(* PLC project Robin, CODESYS CODESYS V3.5 SP15, author pdcribeiro *)
(* stored: creationDateTime 2019-12-17T11:46:08.0055698, version 0.1.2, modificationDateTime 2019-12-17T11:45:59.136833, organization INESC TEC *)
(* A ROS-CODESYS shared memory bridge that maps CODESYS variables to ROS topics.

https://github.com/ScalABLE40/robin *)

(* {attribute 'pack_mode' := '0'} *)
TYPE Accel : STRUCT
  linear : Vector3;
  angular : Vector3;
END_STRUCT;
END_TYPE

(* {attribute 'pack_mode' := '0'} *)
TYPE AccelStamped : STRUCT
  header : Header;
  accel : Accel;
END_STRUCT;
END_TYPE

(* {attribute 'pack_mode' := '0'} *)
TYPE AccelWithCovariance : STRUCT
  accel : Accel;
  covariance : ARRAY[1..36] OF LREAL;
END_STRUCT;
END_TYPE

(* {attribute 'pack_mode' := '0'} *)
TYPE AccelWithCovarianceStamped : STRUCT
  header : Header;
  accel : AccelWithCovariance;
END_STRUCT;
END_TYPE

(* {attribute 'pack_mode' := '0'} *)
TYPE Inertia : STRUCT
  m : LREAL;
  com : Vector3;
  ixx : LREAL;
  ixy : LREAL;
  ixz : LREAL;
  iyy : LREAL;
  iyz : LREAL;
  izz : LREAL;
END_STRUCT;
END_TYPE

(* {attribute 'pack_mode' := '0'} *)
TYPE InertiaStamped : STRUCT
  header : Header;
  inertia : Inertia;
END_STRUCT;
END_TYPE

(* /{attribute 'pack_mode' := '0'} *)
TYPE Point : STRUCT
  x : LREAL;
  y : LREAL;
  z : LREAL;
END_STRUCT;
END_TYPE

(* {attribute 'pack_mode' := '0'} *)
TYPE Point32 : STRUCT
  x : REAL;
  y : REAL;
  z : REAL;
END_STRUCT;
END_TYPE

(* {attribute 'pack_mode' := '0'} *)
TYPE PointStamped : STRUCT
  header : Header;
  point : Point;
END_STRUCT;
END_TYPE

(* {attribute 'pack_mode' := '0'} *)
TYPE Polygon : STRUCT
  {attribute 'robin_var_len'}
  points : ARRAY[1..Robin.DEF_ARRAY_LEN] OF Point32;
END_STRUCT;
END_TYPE

(* {attribute 'pack_mode' := '0'} *)
TYPE PolygonStamped : STRUCT
  header : Header;
  polygon : Polygon;
END_STRUCT;
END_TYPE

(* {attribute 'pack_mode' := '0'} *)
TYPE Pose : STRUCT
  position : Point;
  orientation : Quaternion;
END_STRUCT;
END_TYPE

(* {attribute 'pack_mode' := '0'} *)
TYPE Pose2D : STRUCT
  x : LREAL;
  y : LREAL;
  theta : LREAL;
END_STRUCT;
END_TYPE

(* {attribute 'pack_mode' := '0'} *)
TYPE PoseArray : STRUCT
  header : Header;
  {attribute 'robin_var_len'}
  poses : ARRAY[1..Robin.DEF_ARRAY_LEN] OF Pose;
END_STRUCT;
END_TYPE

(* {attribute 'pack_mode' := '0'} *)
TYPE PoseStamped : STRUCT
  header : Header;
  pose : Pose;
END_STRUCT;
END_TYPE

(* {attribute 'pack_mode' := '0'} *)
TYPE PoseWithCovariance : STRUCT
  pose : Pose;
  covariance : ARRAY[1..36] OF LREAL;
END_STRUCT;
END_TYPE

(* {attribute 'pack_mode' := '0'} *)
TYPE PoseWithCovarianceStamped : STRUCT
  header : Header;
  pose : PoseWithCovariance;
END_STRUCT;
END_TYPE

(* {attribute 'pack_mode' := '0'} *)
TYPE Quaternion : STRUCT
  x : LREAL;
  y : LREAL;
  z : LREAL;
  w : LREAL;
END_STRUCT;
END_TYPE

(* {attribute 'pack_mode' := '0'} *)
TYPE QuaternionStamped : STRUCT
  header : Header;
  quaternion : Quaternion;
END_STRUCT;
END_TYPE

(* {attribute 'pack_mode' := '0'} *)
TYPE Transform : STRUCT
  translation : Vector3;
  rotation : Quaternion;
END_STRUCT;
END_TYPE

(* {attribute 'pack_mode' := '0'} *)
TYPE TransformStamped : STRUCT
  header : Header;
  child_frame_id : STRING;
  transform : Transform;
END_STRUCT;
END_TYPE

(* {attribute 'pack_mode' := '0'} *)
TYPE Twist : STRUCT
  linear : Vector3;
  angular : Vector3;
END_STRUCT;
END_TYPE

(* {attribute 'pack_mode' := '0'} *)
TYPE TwistStamped : STRUCT
  header : Header;
  twist : Twist;
END_STRUCT;
END_TYPE

(* {attribute 'pack_mode' := '0'} *)
TYPE TwistWithCovariance : STRUCT
  twist : Twist;
  covariance : ARRAY[1..Robin.DEF_ARRAY_LEN] OF LREAL;
END_STRUCT;
END_TYPE

(* {attribute 'pack_mode' := '0'} *)
TYPE TwistWithCovarianceStamped : STRUCT
  header : Header;
  twist : TwistWithCovariance;
END_STRUCT;
END_TYPE

(* {attribute 'pack_mode' := '0'} *)
TYPE Vector3 : STRUCT
  x : LREAL;
  y : LREAL;
  z : LREAL;
END_STRUCT;
END_TYPE

(* {attribute 'pack_mode' := '0'} *)
TYPE Vector3Stamped : STRUCT
  header : Header;
  vector : Vector3;
END_STRUCT;
END_TYPE

(* {attribute 'pack_mode' := '0'} *)
TYPE Wrench : STRUCT
  force : Vector3;
  torque : Vector3;
END_STRUCT;
END_TYPE

(* {attribute 'pack_mode' := '0'} *)
TYPE WrenchStamped : STRUCT
  header : Header;
  wrench : Wrench;
END_STRUCT;
END_TYPE

TYPE RobinData : STRUCT
  sem : RTS_IEC_HANDLE;
  shm : RTS_IEC_HANDLE;
  result : RTS_IEC_RESULT;
  bytes : __UXINT;
END_STRUCT;
END_TYPE

TYPE ROS_BOOL : USINT;
END_TYPE

(* deprecated *)
TYPE ROS_BYTE : SINT;
END_TYPE

(* deprecated *)
TYPE ROS_CHAR : USINT;
END_TYPE

(* {attribute 'pack_mode' := '0'} *)
TYPE ROS_DURATION : STRUCT
  secs : UDINT;
  nsecs : UDINT;
END_STRUCT;
END_TYPE

(* {attribute 'pack_mode' := '0'} *)
TYPE ROS_TIME : STRUCT
  secs : UDINT;
  nsecs : UDINT;
END_STRUCT;
END_TYPE

{attribute 'suffixed'}
TYPE Bool_ : STRUCT
  data : BOOL;
END_STRUCT;
END_TYPE

{attribute 'suffixed'}
TYPE Byte_ : STRUCT
  data : BYTE;
END_STRUCT;
END_TYPE

(* {attribute 'pack_mode' := '0'} *)
TYPE ByteMultiArray : STRUCT
  layout : MultiArrayLayout;
  {attribute 'robin_var_len'}
  data : ARRAY[1..Robin.DEF_ARRAY_LEN] OF BYTE;
END_STRUCT;
END_TYPE

TYPE Char : STRUCT
  data : CHAR;
END_STRUCT;
END_TYPE

TYPE ColorRGBA : STRUCT
  {attribute 'suffixed'}
  r_ : REAL;
  g : REAL;
  b : REAL;
  a : REAL;
END_STRUCT;
END_TYPE

TYPE Duration : STRUCT
  data : ROS_DURATION;
END_STRUCT;
END_TYPE

TYPE Float32 : STRUCT
  data : REAL;
END_STRUCT;
END_TYPE

TYPE Float64 : STRUCT
  data : LREAL;
END_STRUCT;
END_TYPE

(* {attribute 'pack_mode' := '0'} *)
TYPE Header : STRUCT
  seq : UDINT;
  stamp : ROS_TIME;
  frame_id : STRING(83);
END_STRUCT;
END_TYPE

TYPE Int16 : STRUCT
  data : INT;
END_STRUCT;
END_TYPE

(* {attribute 'pack_mode' := '0'} *)
TYPE Int16MultiArray : STRUCT
  layout : MultiArrayLayout;
  {attribute 'robin_var_len'}
  data : ARRAY[1..Robin.DEF_ARRAY_LEN] OF INT;
END_STRUCT;
END_TYPE

TYPE Int32 : STRUCT
  data : DINT;
END_STRUCT;
END_TYPE

(* {attribute 'pack_mode' := '0'} *)
TYPE Int32MultiArray : STRUCT
  layout : MultiArrayLayout;
  {attribute 'robin_var_len'}
  data : ARRAY[1..Robin.DEF_ARRAY_LEN] OF DINT;
END_STRUCT;
END_TYPE

TYPE Int64 : STRUCT
  data : LINT;
END_STRUCT;
END_TYPE

(* {attribute 'pack_mode' := '0'} *)
TYPE Int64MultiArray : STRUCT
  layout : MultiArrayLayout;
  {attribute 'robin_var_len'}
  data : ARRAY[1..Robin.DEF_ARRAY_LEN] OF LINT;
END_STRUCT;
END_TYPE

TYPE Int8 : STRUCT
  data : SINT;
END_STRUCT;
END_TYPE

(* {attribute 'pack_mode' := '0'} *)
TYPE Int8MultiArray : STRUCT
  layout : MultiArrayLayout;
  {attribute 'robin_var_len'}
  data : ARRAY[1..Robin.DEF_ARRAY_LEN] OF SINT;
END_STRUCT;
END_TYPE

(* {attribute 'pack_mode' := '0'} *)
TYPE MultiArrayDimension : STRUCT
  label : STRING;
  size : UDINT;
  stride : UDINT;
END_STRUCT;
END_TYPE

(* /{attribute 'pack_mode' := '0'} *)
TYPE MultiArrayLayout : STRUCT
  {attribute 'robin_var_len'}
  dim : ARRAY[1..Robin.DEF_ARRAY_LEN] OF MultiArrayDimension;
  data_offset : UDINT;
END_STRUCT;
END_TYPE

{attribute 'suffixed'}
TYPE String_ : STRUCT
  data : STRING;
END_STRUCT;
END_TYPE

{attribute 'suffixed'}
TYPE Time_ : STRUCT
  data : ROS_TIME;
END_STRUCT;
END_TYPE

TYPE UInt16 : STRUCT
  data : UINT;
END_STRUCT;
END_TYPE

(* {attribute 'pack_mode' := '0'} *)
TYPE UInt16MultiArray : STRUCT
  layout : MultiArrayLayout;
  {attribute 'robin_var_len'}
  data : ARRAY[1..Robin.DEF_ARRAY_LEN] OF UINT;
END_STRUCT;
END_TYPE

TYPE UInt32 : STRUCT
  data : UDINT;
END_STRUCT;
END_TYPE

(* {attribute 'pack_mode' := '0'} *)
TYPE UInt32MultiArray : STRUCT
  layout : MultiArrayLayout;
  {attribute 'robin_var_len'}
  data : ARRAY[1..Robin.DEF_ARRAY_LEN] OF UDINT;
END_STRUCT;
END_TYPE

TYPE UInt64 : STRUCT
  data : ULINT;
END_STRUCT;
END_TYPE

(* {attribute 'pack_mode' := '0'} *)
TYPE UInt64MultiArray : STRUCT
  layout : MultiArrayLayout;
  {attribute 'robin_var_len'}
  data : ARRAY[1..Robin.DEF_ARRAY_LEN] OF ULINT;
END_STRUCT;
END_TYPE

TYPE UInt8 : STRUCT
  data : USINT;
END_STRUCT;
END_TYPE

(* {attribute 'pack_mode' := '0'} *)
TYPE UInt8MultiArray : STRUCT
  layout : MultiArrayLayout;
  {attribute 'robin_var_len'}
  data : ARRAY[1..Robin.DEF_ARRAY_LEN] OF USINT;
END_STRUCT;
END_TYPE

(* {attribute 'pack_mode' := '0'} *)
TYPE BatteryState : STRUCT
  header : Header;
  voltage : REAL;
  current : REAL;
  charge : REAL;
  capacity : REAL;
  design_capacity : REAL;
  percentage : REAL;
  power_supply_status : USINT;
  power_supply_health : USINT;
  power_supply_technology : USINT;
  present : BOOL;
  {attribute 'robin_var_len'}
  cell_voltage : ARRAY[1..Robin.DEF_ARRAY_LEN] OF REAL;
  location : STRING;
  serial_number : STRING;
END_STRUCT;
END_TYPE

(* {attribute 'pack_mode' := '0'} *)
TYPE CameraInfo : STRUCT
  header : Header;
  height : UDINT;
  width : UDINT;
  distortion_model : STRING;
  {attribute 'robin_var_len'}
  D : ARRAY[1..Robin.DEF_ARRAY_LEN] OF LREAL;
  K : ARRAY[1..9] OF LREAL;
  R : ARRAY[1..9] OF LREAL;
  P : ARRAY[1..12] OF LREAL;
  binning_x : UDINT;
  binning_y : UDINT;
  roi : RegionOfInterest;
END_STRUCT;
END_TYPE

(* {attribute 'pack_mode' := '0'} *)
TYPE ChannelFloat32 : STRUCT
  name : STRING;
  {attribute 'robin_var_len'}
  values : ARRAY[1..Robin.DEF_ARRAY_LEN] OF REAL;
END_STRUCT;
END_TYPE

(* {attribute 'pack_mode' := '0'} *)
TYPE CompressedImage : STRUCT
  header : Header;
  format : STRING;
  {attribute 'robin_var_len'}
  data : ARRAY[1..Robin.DEF_ARRAY_LEN] OF USINT;
END_STRUCT;
END_TYPE

(* {attribute 'pack_mode' := '0'} *)
TYPE FluidPressure : STRUCT
  header : Header;
  fluid_pressure : LREAL;
  variance : LREAL;
END_STRUCT;
END_TYPE

(* {attribute 'pack_mode' := '0'} *)
TYPE Illuminance : STRUCT
  header : Header;
  illuminance : LREAL;
  variance : LREAL;
END_STRUCT;
END_TYPE

(* {attribute 'pack_mode' := '0'} *)
TYPE Image : STRUCT
  header : Header;
  height : UDINT;
  width : UDINT;
  encoding : STRING;
  is_bigendian : USINT;
  step : UDINT;
  {attribute 'robin_var_len'}
  data : ARRAY[1..Robin.DEF_ARRAY_LEN] OF USINT;
END_STRUCT;
END_TYPE

(* {attribute 'pack_mode' := '0'} *)
TYPE Imu : STRUCT
  header : Header;
  orientation : Quaternion;
  orientation_covariance : ARRAY[1..9] OF LREAL;
  angular_velocity : Vector3;
  angular_velocity_covariance : ARRAY[1..9] OF LREAL;
  linear_acceleration : Vector3;
  linear_acceleration_covariance : ARRAY[1..9] OF LREAL;
END_STRUCT;
END_TYPE

(* {attribute 'pack_mode' := '0'} *)
TYPE JointState : STRUCT
  header : Header;
  {attribute 'robin_var_len'}
  name : ARRAY[1..Robin.DEF_ARRAY_LEN] OF STRING;
  {attribute 'robin_var_len'}
  position : ARRAY[1..Robin.DEF_ARRAY_LEN] OF LREAL;
  {attribute 'robin_var_len'}
  velocity : ARRAY[1..Robin.DEF_ARRAY_LEN] OF LREAL;
  {attribute 'robin_var_len'}
  effort : ARRAY[1..Robin.DEF_ARRAY_LEN] OF LREAL;
END_STRUCT;
END_TYPE

(* {attribute 'pack_mode' := '0'} *)
TYPE Joy : STRUCT
  header : Header;
  {attribute 'robin_var_len'}
  axes : ARRAY[1..Robin.DEF_ARRAY_LEN] OF REAL;
  {attribute 'robin_var_len'}
  buttons : ARRAY[1..Robin.DEF_ARRAY_LEN] OF DINT;
END_STRUCT;
END_TYPE

(* {attribute 'pack_mode' := '0'} *)
TYPE JoyFeedback : STRUCT
  type : USINT;
  id : USINT;
  intensity : REAL;
END_STRUCT;
END_TYPE

(* {attribute 'pack_mode' := '0'} *)
TYPE JoyFeedbackArray : STRUCT
  {attribute 'robin_var_len'}
  array : ARRAY[1..Robin.DEF_ARRAY_LEN] OF JoyFeedback;
END_STRUCT;
END_TYPE

(* {attribute 'pack_mode' := '0'} *)
TYPE LaserEcho : STRUCT
  {attribute 'robin_var_len'}
  echoes : ARRAY[1..Robin.DEF_ARRAY_LEN] OF REAL;
END_STRUCT;
END_TYPE

(* {attribute 'pack_mode' := '0'} *)
TYPE LaserScan : STRUCT
  header : Header;
  angle_min : REAL;
  angle_max : REAL;
  angle_increment : REAL;
  time_increment : REAL;
  scan_time : REAL;
  range_min : REAL;
  range_max : REAL;
  {attribute 'robin_var_len'}
  ranges : ARRAY[1..Robin.DEF_ARRAY_LEN] OF REAL;
  {attribute 'robin_var_len'}
  intensities : ARRAY[1..Robin.DEF_ARRAY_LEN] OF REAL;
END_STRUCT;
END_TYPE

(* {attribute 'pack_mode' := '0'} *)
TYPE MagneticField : STRUCT
  header : Header;
  magnetic_field : Vector3;
  intensities : ARRAY[1..9] OF REAL;
END_STRUCT;
END_TYPE

(* {attribute 'pack_mode' := '0'} *)
TYPE MultiDOFJointState : STRUCT
  header : Header;
  {attribute 'robin_var_len'}
  joint_names : ARRAY[1..Robin.DEF_ARRAY_LEN] OF STRING;
  {attribute 'robin_var_len'}
  transforms : ARRAY[1..Robin.DEF_ARRAY_LEN] OF Transform;
  {attribute 'robin_var_len'}
  twist : ARRAY[1..Robin.DEF_ARRAY_LEN] OF Twist;
  {attribute 'robin_var_len'}
  wrench : ARRAY[1..Robin.DEF_ARRAY_LEN] OF Wrench;
END_STRUCT;
END_TYPE

(* {attribute 'pack_mode' := '0'} *)
TYPE MultiEchoLaserScan : STRUCT
  header : Header;
  angle_min : REAL;
  angle_max : REAL;
  angle_increment : REAL;
  time_increment : REAL;
  scan_time : REAL;
  range_min : REAL;
  range_max : REAL;
  {attribute 'robin_var_len'}
  ranges : ARRAY[1..Robin.DEF_ARRAY_LEN] OF LaserEcho;
  {attribute 'robin_var_len'}
  intensities : ARRAY[1..Robin.DEF_ARRAY_LEN] OF LaserEcho;
END_STRUCT;
END_TYPE

(* {attribute 'pack_mode' := '0'} *)
TYPE NavSatFix : STRUCT
  header : Header;
  status : NavSatStatus;
  latitude : LREAL;
  longitude : LREAL;
  altitude : LREAL;
  position_covariance : ARRAY[1..9] OF LREAL;
  position_covariance_type : USINT;
END_STRUCT;
END_TYPE

(* {attribute 'pack_mode' := '0'} *)
TYPE NavSatStatus : STRUCT
  status : SINT;
  service : UINT;
END_STRUCT;
END_TYPE

(* {attribute 'pack_mode' := '0'} *)
TYPE PointCloud : STRUCT
  header : Header;
  {attribute 'robin_var_len'}
  points : ARRAY[1..Robin.DEF_ARRAY_LEN] OF Point32;
  {attribute 'robin_var_len'}
  channels : ARRAY[1..Robin.DEF_ARRAY_LEN] OF ChannelFloat32;
END_STRUCT;
END_TYPE

(* {attribute 'pack_mode' := '0'} *)
TYPE PointCloud2 : STRUCT
  header : Header;
  height : UDINT;
  width : UDINT;
  {attribute 'robin_var_len'}
  fields : ARRAY[1..Robin.DEF_ARRAY_LEN] OF PointField;
  is_bigendian : BOOL;
  point_step : UDINT;
  row_step : UDINT;
  {attribute 'robin_var_len'}
  data : ARRAY[1..Robin.DEF_ARRAY_LEN] OF USINT;
  is_dense : BOOL;
END_STRUCT;
END_TYPE

(* {attribute 'pack_mode' := '0'} *)
TYPE PointField : STRUCT
  name : STRING;
  offset : UDINT;
  datatype : USINT;
  count : UDINT;
END_STRUCT;
END_TYPE

(* {attribute 'pack_mode' := '0'} *)
TYPE Range : STRUCT
  header : ?;
  radiation_type : USINT;
  field_of_view : REAL;
  min_range : REAL;
  max_range : REAL;
  range : REAL;
END_STRUCT;
END_TYPE

(* {attribute 'pack_mode' := '0'} *)
TYPE RegionOfInterest : STRUCT
  x_offset : UDINT;
  y_offset : UDINT;
  height : UDINT;
  width : UDINT;
  do_rectify : BOOL;
END_STRUCT;
END_TYPE

(* {attribute 'pack_mode' := '0'} *)
TYPE RelativeHumidity : STRUCT
  header : ?;
  relative_humidity : LREAL;
  variance : LREAL;
END_STRUCT;
END_TYPE

(* {attribute 'pack_mode' := '0'} *)
TYPE Temperature : STRUCT
  header : ?;
  temperature : LREAL;
  variance : LREAL;
END_STRUCT;
END_TYPE

(* {attribute 'pack_mode' := '0'} *)
TYPE TimeReference : STRUCT
  header : ?;
  time_ref : ROS_TIME;
  source : STRING;
END_STRUCT;
END_TYPE

FUNCTION_BLOCK Robin
  VAR CONSTANT
    MAX_SIZE : INT := 20;
    SEM_TIMEOUT : UDINT := 1000;  (* in ms (16#FFFFFFFF = inf) *)
  END_VAR
  VAR_OUTPUT CONSTANT
    DEF_ARRAY_LEN : INT := 20;
  END_VAR
  VAR
    data : ARRAY[1..MAX_SIZE] OF RobinData;
    idx : UINT;
    i : INT;
  END_VAR

            idx := 1;

          

(* FB_Init is always available implicitly and it is used primarily for initialization. The return value is not evaluated. For a specific influence, you can also declare the methods explicitly and provide additional code there with the standard initialization code. You can evaluate the return value. *)
METHOD FB_Init : BOOL
  VAR_INPUT
    bInitRetains : BOOL;  (* TRUE: the retain variables are initialized (reset warm / reset cold) *)
    bInCopyCode : BOOL;  (* TRUE: the instance will be copied to the copy code afterward (online change) *)
  END_VAR
                  FOR i := 1 TO MAX_SIZE DO
	data[i].sem := RTS_INVALID_HANDLE;
	data[i].shm := RTS_INVALID_HANDLE;
END_FOR;

                
END_METHOD

(* FB_Exit must be implemented explicitly. If there is an implementation, then the method is called before the controller removes the code of the function block instance (implicit call). The return value is not evaluated. *)
METHOD FB_Exit : BOOL
  VAR_INPUT
    bInCopyCode : BOOL;  (* TRUE: the exit method is called in order to leave the instance which will be copied afterwards (online change). *)
  END_VAR
                  // IF NOT bInCopyCode THEN
// 	result := SysSemProcessEnter(sem, SEM_TIMEOUT);
	FOR i := 1 TO MAX_SIZE DO
		IF data[idx].shm <> RTS_INVALID_HANDLE THEN
			data[idx].result := SysSharedMemoryClose(data[idx].shm);
// 			data[idx].result := SysSharedMemoryDelete(data[idx].shm);
		END_IF
	END_FOR;
// 	result := SysSharedMemoryDelete(shm);
// 	result := SysSemProcessDelete(sem);
// END_IF

                
END_METHOD

METHOD open : BOOL
  VAR_INPUT
    name : STRING;
    size : __UXINT;
  END_VAR
                  IF data[idx].shm = RTS_INVALID_HANDLE THEN
	data[idx].shm := SysSharedMemoryOpen2(name, 0, ADR(size), ADR(data[idx].result));
	IF data[idx].shm <> RTS_INVALID_HANDLE THEN
		data[idx].sem := SysSemProcessCreate(name, ADR(data[idx].result));
		IF data[idx].sem <> RTS_INVALID_HANDLE THEN
			open := TRUE;
		ELSE
			open := FALSE;
		END_IF
	ELSE
		open := FALSE;
	END_IF
ELSE
	open := TRUE;
END_IF

                
END_METHOD

{attribute 'hasanytype'}
METHOD read
  VAR_INPUT
    name : STRING;
    {attribute 'anytypeclass' := 'ANY'}
    var_ : __SYSTEM.AnyType;
  END_VAR
  VAR
    size : __UXINT := DINT_TO___UXINT(var_.diSize);
  END_VAR
                  IF open(name, size) THEN
	IF SysSemProcessEnter(data[idx].sem, SEM_TIMEOUT) = Errors.ERR_OK THEN
		data[idx].bytes := SysSharedMemoryRead(data[idx].shm, 0, var_.pValue, size, ADR(data[idx].result));
		data[idx].result := SysSemProcessLeave(data[idx].sem);
	END_IF
END_IF
idx := idx + 1;

                
END_METHOD

{attribute 'hasanytype'}
METHOD write
  VAR_INPUT
    name : STRING;
    {attribute 'anytypeclass' := 'ANY'}
    var_ : __SYSTEM.AnyType;
  END_VAR
  VAR
    size : __UXINT := DINT_TO___UXINT(var_.diSize);
  END_VAR
                  IF open(name, size) THEN
	IF SysSemProcessEnter(data[idx].sem, SEM_TIMEOUT) = Errors.ERR_OK THEN
		data[idx].bytes := SysSharedMemoryWrite(data[idx].shm, 0, var_.pValue, size, ADR(data[idx].result));
		data[idx].result := SysSemProcessLeave(data[idx].sem);
	END_IF
END_IF
idx := idx + 1;

                
END_METHOD
END_FUNCTION_BLOCK
